PROGRAM MAIN
VAR
END_VAR

END_PROGRAM

(* stored: Version 1.1.0.1
   POU MAIN: Id {6692eb13-f07c-4d90-a32e-02009e09e61b} *)
